TYPE FsT_VarInfo : __SYSTEM.VAR_INFO; END_TYPE

(* stored: Version 1.1.0.1, ProductVersion 3.1.4024.4
   DUT FsT_VarInfo: Id {7f640f5f-c9d5-43fc-8cca-faed761122ae} *)
